FUNCTION_BLOCK Vehiculo IMPLEMENTS I_Mover


METHOD Mover : REAL
VAR_INPUT
	Velocidad_Deseada : REAL;
END_VAR
Mover := Velocidad_Deseada;
END_METHOD

END_FUNCTION_BLOCK

(* stored: Version 1.1.0.1, ProductVersion 3.1.4024.12
   POU Vehiculo: Id {d9f89bc7-2a9b-4dca-a00a-6ec7dcda740f}, SpecialFunc None
   Method Mover: Id {e36f3dcf-1ae2-4c88-a575-1852fbfc4d20} *)
